# EPICS substitutions: ek9000App/Db/EL4021.substitutions
file EL4021.template
{       pattern
        {
                TERMINAL,

        }
        {
        }
}
